TYPE S_General :
STRUCT
	Full_speed: REAL;
	Slow_switch_speed: REAL;
	Creep_switch_speed: REAL;
	Enforced_slow_speed: REAL;
	Clutch_out_Speed: REAL;
	Rope_capping_speed: REAL;
	Slinging_speed: REAL;
	Speed_ramp_rate: REAL;
	Speed_s_curve_ms: REAL;
	Current_limit: REAL;
	Brake_test_current: REAL;
	Full_lever_amps: REAL;
END_STRUCT
END_TYPE

(* stored: Version 1.1.0.1, ProductVersion 3.1.4024.0
   DUT S_General: Id {dac1af7d-f143-4f63-acd2-b3e2b45ad630} *)
